FUNCTION_BLOCK ServiceInterface (* Service Interface Function Block Type *)
  (* Standard: 61499-2 *)
  (* Version 0.0, 2008-07-10, 4DIAC-IDE, 4DIAC-Consortium *)
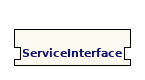
END_FUNCTION_BLOCK
